(* CODESYS project SheetMetalFactoryLib.library
   Version: 0.0.0.1
   Author: RDOE
   Title: Sheet Metal Factory
   Description: Example Library to make use of FB Factory based on template provided with standard library project from wizard
   Placeholder: PlaceholderTemplate
   DocFormat: reStructuredText
   DefaultNamespace: SMF
   LanguageModelAttribute: qualified-access-only
   Company: OSB AG

Project tree, tasks and I/O mapping:
  libraries: CAA Types Extern, * (CAA Technical Workgroup); CAA Behaviour Model, * (CAA Technical Workgroup); CAA FB Factory, * (CAA Technical Workgroup)
  SheetMetalFactoryLib/
    Enums/
      data type ERROR
      data type WorkerDataType
      data type STATE
    Function Blocks/
      function block WorkerFactory [ST]: createIdle, prvInstCount, prvInstPoolExtendsFactor, prvInstSize, createCutter, createPolisher, createWorker
      function block ProcessController [ST]: FB_INIT
      Cutter/
        function block Cutter [ST]: init, prvInstInit, cutEdge, getState, setState, workerType, process, nextWorker, setNextWorker
        function block CutterData [ST]: workerType
      Polisher/
        function block Polisher [ST]: init, prvInstInit, polish, getState, setState, workerType, process, nextWorker, setNextWorker
        function block PolisherData [ST]: workerType
      Idle/
        function block Idle [ST]: setState, prvInstInit, nextWorker, workerType, process, setNextWorker
        function block IdleData [ST]: workerType
      function block SequenceFactory [ST]: FB_INIT, generateSequence, cleanUp
    Functions/
      Helper/
        function decrementInt [ST]
        function incrementInt [ST]
    GlobalConstants/
      global variables Constants
    GlobalVariables/
      global variables Variables
    Interfaces/
      interface IWorkerData: workerType
      interface IWorker: workerType, process, nextWorker, setNextWorker
    Structs/
    Templates/
      Behaviour Model/
        function block ETrigA_Temp [ST]: prvAbort, prvCyclicAction, prvResetOutputs, prvStart
        function block ETrigTlA_Temp [ST]: prvAbort, prvCyclicAction, prvResetOutputs, prvStart
        function block ETrigTl_Temp [ST]: prvAbort, prvCyclicAction, prvResetOutputs, prvStart
        function block ETrigToA_Temp [ST]: prvAbort, prvCyclicAction, prvResetOutputs, prvStart
        function block ETrigToTlA_Temp [ST]: prvAbort, prvCyclicAction, prvResetOutputs, prvStart
        function block ETrigToTl_Temp [ST]: prvAbort, prvCyclicAction, prvResetOutputs, prvStart
        function block ETrigTo_Temp [ST]: prvAbort, prvCyclicAction, prvResetOutputs, prvStart
        function block ETrig_Temp [ST]: prvAbort, prvCyclicAction, prvResetOutputs, prvStart
        function block LTrig_Temp [ST]: prvAbort, prvCyclicAction, prvResetOutputs, prvStart
      FB Factory/
        function block CustomData [ST]
        function block CustomFB [ST]: prvInstInit
        function block CustomFBFactory_heap [ST]: Create, prvInstCount, prvInstPoolExtendsFactor, prvInstSize
        function block CustomFBFactory_static [ST]: Create, prvInstPoolAdr, prvInstPoolSize, prvInstSize
    Types/
*)

// SheetMetalFactoryLib/Enums/ERROR
{attribute 'qualified_only'}
//{attribute 'conditionalshow'}
//{attribute 'conditionalshow' := 'SomeText'}
//{attribute 'hide'}
TYPE ERROR : 
(
	NO_ERROR := 0, 
	TIME_OUT
); 
END_TYPE

// SheetMetalFactoryLib/Enums/WorkerDataType
{attribute 'qualified_only'}
{attribute 'strict'}
TYPE WorkerDataType :
(
	NotSpecified :=-1,
	Idle := 0,
	Cutter,
	Polisher,
	Engraver
) := NotSpecified;
END_TYPE

// SheetMetalFactoryLib/Enums/STATE
{attribute 'qualified_only'}
{attribute 'strict'}
TYPE STATE :
(
	idle := 0,
	firstEdge,
	secondEdge,
	thirdEdge,
	fourthEdge,
	done,
	error := -1
	
);
END_TYPE

// SheetMetalFactoryLib/GlobalConstants/Constants
{attribute 'qualified_only'}
//{attribute 'conditionalshow'}
//{attribute 'conditionalshow' := 'SomeText'}
//{attribute 'hide'}
VAR_GLOBAL CONSTANT
	gc_iDummy : INT := 42; /// This is a dummy global constant variable
END_VAR

// SheetMetalFactoryLib/GlobalVariables/Variables
{attribute 'qualified_only'}
//{attribute 'conditionalshow'}
//{attribute 'conditionalshow' := 'SomeText'}
//{attribute 'hide'}
VAR_GLOBAL
	g_iDummy : INT; /// This is a dummy global variable
END_VAR

// SheetMetalFactoryLib/Templates/Behaviour Model/ETrigA_Temp
//{attribute 'hide_all_locals'}
//{attribute 'conditionalshow_all_locals' := 'SomeText'}
//{attribute 'conditionalshow_all_locals'}
//{attribute 'conditionalshow' := 'SomeText'}
//{attribute 'conditionalshow'}
//{attribute 'hide'}
FUNCTION_BLOCK ETrigA_Temp EXTENDS CBM.ETrigA
VAR_INPUT
	(* specific Inputs *)
END_VAR
VAR_OUTPUT
	eError : ERROR;
	(* specific Outputs *)
END_VAR
VAR
	(* specific vars *)
END_VAR

SUPER^();
IF iError = CBM.ERROR.TIME_OUT THEN
	eError := ERROR.TIME_OUT;
ELSE
	eError := iError;
END_IF

{attribute 'hide'}
METHOD prvAbort : BOOL
VAR_INPUT
END_VAR
VAR
END_VAR
IF xError THEN (* abort because of error *)
	(* TODO: insert specific Code here *)
ELSE (* user abort *)
	(* TODO: insert specific Code here *)
END_IF
xAbortInProgress:= FALSE;
END_METHOD

{attribute 'hide'}
METHOD prvCyclicAction : BOOL
VAR_INPUT
END_VAR
VAR
END_VAR
(* TODO: insert specific Code here *)
xDone:= TRUE;
(* if an error occurs, set iError to a value else than zero instead of xDone:= TRUE *)
(* to keep repeat loop *)
END_METHOD

{attribute 'hide'}
METHOD prvResetOutputs : BOOL
VAR_INPUT
END_VAR
VAR
END_VAR
(* TODO: insert specific Code here *)
SUPER^.prvResetOutputs();
END_METHOD

{attribute 'hide'}
METHOD prvStart : BOOL
VAR_INPUT
END_VAR
VAR
END_VAR
(* this code is called, when the application is started (rising edge of xExecute *)
(* TODO: copy specific input variables into local copies *)
(* TODO: insert specific Code here *)
;
END_METHOD

END_FUNCTION_BLOCK

// SheetMetalFactoryLib/Templates/Behaviour Model/ETrigTlA_Temp
//{attribute 'hide_all_locals'}
//{attribute 'conditionalshow_all_locals' := 'SomeText'}
//{attribute 'conditionalshow_all_locals'}
//{attribute 'conditionalshow' := 'SomeText'}
//{attribute 'conditionalshow'}
//{attribute 'hide'}
FUNCTION_BLOCK ETrigTlA_Temp EXTENDS CBM.ETrigTlA
VAR_INPUT
	(* specific Inputs *)
END_VAR
VAR_OUTPUT
	eError : ERROR;
	(* specific Outputs *)
END_VAR
VAR
	(* specific vars *)
END_VAR

SUPER^();
IF iError = CBM.ERROR.TIME_OUT THEN
	eError := ERROR.TIME_OUT;
ELSE
	eError := iError;
END_IF

{attribute 'hide'}
METHOD prvAbort : BOOL
VAR_INPUT
END_VAR
VAR
END_VAR
IF xError THEN (* abort because of error *)
	(* TODO: insert specific Code here *)
ELSE (* user abort *)
	(* TODO: insert specific Code here *)
END_IF
xAbortInProgress:= FALSE;
END_METHOD

{attribute 'hide'}
METHOD prvCyclicAction : BOOL
VAR_INPUT
END_VAR
VAR
END_VAR
(* TODO: insert specific Code here *)
xDone:= TRUE;
(* if an error occurs, set iError to a value else than zero instead of xDone:= TRUE *)
(* to keep repeat loop *)
END_METHOD

{attribute 'hide'}
METHOD prvResetOutputs : BOOL
VAR_INPUT
END_VAR
VAR
END_VAR
(* TODO: insert specific Code here *)
SUPER^.prvResetOutputs();
END_METHOD

{attribute 'hide'}
METHOD prvStart : BOOL
VAR_INPUT
END_VAR
VAR
END_VAR
(* this code is called, when the application is started (rising edge of xExecute *)
(* TODO: copy specific input variables into local copies *)
(* TODO: insert specific Code here *)
;
END_METHOD

END_FUNCTION_BLOCK

// SheetMetalFactoryLib/Templates/Behaviour Model/ETrigTl_Temp
//{attribute 'hide_all_locals'}
//{attribute 'conditionalshow_all_locals' := 'SomeText'}
//{attribute 'conditionalshow_all_locals'}
//{attribute 'conditionalshow' := 'SomeText'}
//{attribute 'conditionalshow'}
//{attribute 'hide'}
FUNCTION_BLOCK ETrigA_Temp EXTENDS CBM.ETrigTl
VAR_INPUT
	(* specific Inputs *)
END_VAR
VAR_OUTPUT
	eError : ERROR;
	(* specific Outputs *)
END_VAR
VAR
	(* specific vars *)
END_VAR

SUPER^();
IF iError = CBM.ERROR.TIME_OUT THEN
	eError := ERROR.TIME_OUT;
ELSE
	eError := iError;
END_IF

{attribute 'hide'}
METHOD prvAbort : BOOL
VAR_INPUT
END_VAR
VAR
END_VAR
IF xError THEN (* abort because of error *)
	(* TODO: insert specific Code here *)
ELSE (* user abort *)
	(* TODO: insert specific Code here *)
END_IF
xAbortInProgress:= FALSE;
END_METHOD

{attribute 'hide'}
METHOD prvCyclicAction : BOOL
VAR_INPUT
END_VAR
VAR
END_VAR
(* TODO: insert specific Code here *)
xDone:= TRUE;
(* if an error occurs, set iError to a value else than zero instead of xDone:= TRUE *)
(* to keep repeat loop *)
END_METHOD

{attribute 'hide'}
METHOD prvResetOutputs : BOOL
VAR_INPUT
END_VAR
VAR
END_VAR
(* TODO: insert specific Code here *)
SUPER^.prvResetOutputs();
END_METHOD

{attribute 'hide'}
METHOD prvStart : BOOL
VAR_INPUT
END_VAR
VAR
END_VAR
(* this code is called, when the application is started (rising edge of xExecute *)
(* TODO: copy specific input variables into local copies *)
(* TODO: insert specific Code here *)
;
END_METHOD

END_FUNCTION_BLOCK

// SheetMetalFactoryLib/Templates/Behaviour Model/ETrigToA_Temp
//{attribute 'hide_all_locals'}
//{attribute 'conditionalshow_all_locals' := 'SomeText'}
//{attribute 'conditionalshow_all_locals'}
//{attribute 'conditionalshow' := 'SomeText'}
//{attribute 'conditionalshow'}
//{attribute 'hide'}
FUNCTION_BLOCK ETrigToA_Temp EXTENDS CBM.ETrigToA
VAR_INPUT
	(* specific Inputs *)
END_VAR
VAR_OUTPUT
	eError : ERROR;
	(* specific Outputs *)
END_VAR
VAR
	(* specific vars *)
END_VAR

SUPER^();
IF iError = CBM.ERROR.TIME_OUT THEN
	eError := ERROR.TIME_OUT;
ELSE
	eError := iError;
END_IF

{attribute 'hide'}
METHOD prvAbort : BOOL
VAR_INPUT
END_VAR
VAR
END_VAR
IF xError THEN (* abort because of error *)
	(* TODO: insert specific Code here *)
ELSE (* user abort *)
	(* TODO: insert specific Code here *)
END_IF
xAbortInProgress:= FALSE;
END_METHOD

{attribute 'hide'}
METHOD prvCyclicAction : BOOL
VAR_INPUT
END_VAR
VAR
END_VAR
(* TODO: insert specific Code here *)
xDone:= TRUE;
(* if an error occurs, set iError to a value else than zero instead of xDone:= TRUE *)
END_METHOD

{attribute 'hide'}
METHOD prvResetOutputs : BOOL
VAR_INPUT
END_VAR
VAR
END_VAR
(* TODO: insert specific Code here *)
SUPER^.prvResetOutputs();
END_METHOD

{attribute 'hide'}
METHOD prvStart : BOOL
VAR_INPUT
END_VAR
VAR
END_VAR
(* this code is called, when the application is started (rising edge of xExecute *)
(* TODO: copy specific input variables into local copies *)
(* TODO: insert specific Code here *)
;
END_METHOD

END_FUNCTION_BLOCK

// SheetMetalFactoryLib/Templates/Behaviour Model/ETrigToTlA_Temp
//{attribute 'hide_all_locals'}
//{attribute 'conditionalshow_all_locals' := 'SomeText'}
//{attribute 'conditionalshow_all_locals'}
//{attribute 'conditionalshow' := 'SomeText'}
//{attribute 'conditionalshow'}
//{attribute 'hide'}
FUNCTION_BLOCK ETrigToTlA_Temp EXTENDS CBM.ETrigToTlA
VAR_INPUT
	(* specific Inputs *)
END_VAR
VAR_OUTPUT
	eError : ERROR;
	(* specific Outputs *)
END_VAR
VAR
	(* specific vars *)
END_VAR

SUPER^();
IF iError = CBM.ERROR.TIME_OUT THEN
	eError := ERROR.TIME_OUT;
ELSE
	eError := iError;
END_IF

{attribute 'hide'}
METHOD prvAbort : BOOL
VAR_INPUT
END_VAR
VAR
END_VAR
IF xError THEN (* abort because of error *)
	(* TODO: insert specific Code here *)
ELSE (* user abort *)
	(* TODO: insert specific Code here *)
END_IF
xAbortInProgress:= FALSE;
END_METHOD

{attribute 'hide'}
METHOD prvCyclicAction : BOOL
VAR_INPUT
END_VAR
VAR
END_VAR
(* TODO: insert specific Code here *)
xDone:= TRUE;
(* if an error occurs, set iError to a value else than zero instead of xDone:= TRUE *)
(* to keep repeat loop *)
END_METHOD

{attribute 'hide'}
METHOD prvResetOutputs : BOOL
VAR_INPUT
END_VAR
VAR
END_VAR
(* TODO: insert specific Code here *)
SUPER^.prvResetOutputs();
END_METHOD

{attribute 'hide'}
METHOD prvStart : BOOL
VAR_INPUT
END_VAR
VAR
END_VAR
(* this code is called, when the application is started (rising edge of xExecute *)
(* TODO: copy specific input variables into local copies *)
(* TODO: insert specific Code here *)
;
END_METHOD

END_FUNCTION_BLOCK

// SheetMetalFactoryLib/Templates/Behaviour Model/ETrigToTl_Temp
//{attribute 'hide_all_locals'}
//{attribute 'conditionalshow_all_locals' := 'SomeText'}
//{attribute 'conditionalshow_all_locals'}
//{attribute 'conditionalshow' := 'SomeText'}
//{attribute 'conditionalshow'}
//{attribute 'hide'}
FUNCTION_BLOCK ETrigToTl_Temp EXTENDS CBM.ETrigToTl
VAR_INPUT
	(* specific Inputs *)
END_VAR
VAR_OUTPUT
	eError : ERROR;
	(* specific Outputs *)
END_VAR
VAR
	(* specific vars *)
END_VAR

SUPER^();
IF iError = CBM.ERROR.TIME_OUT THEN
	eError := ERROR.TIME_OUT;
ELSE
	eError := iError;
END_IF

{attribute 'hide'}
METHOD prvAbort : BOOL
VAR_INPUT
END_VAR
VAR
END_VAR
IF xError THEN (* abort because of error *)
	(* TODO: insert specific Code here *)
ELSE (* user abort *)
	(* TODO: insert specific Code here *)
END_IF
xAbortInProgress:= FALSE;
END_METHOD

{attribute 'hide'}
METHOD prvCyclicAction : BOOL
VAR_INPUT
END_VAR
VAR
END_VAR
(* TODO: insert specific Code here *)
xDone:= TRUE;
(* if an error occurs, set iError to a value else than zero instead of xDone:= TRUE *)
(* to keep repeat loop *)
END_METHOD

{attribute 'hide'}
METHOD prvResetOutputs : BOOL
VAR_INPUT
END_VAR
VAR
END_VAR
(* TODO: insert specific Code here *)
SUPER^.prvResetOutputs();
END_METHOD

{attribute 'hide'}
METHOD prvStart : BOOL
VAR_INPUT
END_VAR
VAR
END_VAR
(* this code is called, when the application is started (rising edge of xExecute *)
(* TODO: copy specific input variables into local copies *)
(* TODO: insert specific Code here *)
;
END_METHOD

END_FUNCTION_BLOCK

// SheetMetalFactoryLib/Templates/Behaviour Model/ETrigTo_Temp
//{attribute 'hide_all_locals'}
//{attribute 'conditionalshow_all_locals' := 'SomeText'}
//{attribute 'conditionalshow_all_locals'}
//{attribute 'conditionalshow' := 'SomeText'}
//{attribute 'conditionalshow'}
//{attribute 'hide'}
FUNCTION_BLOCK ETrigTo_Temp EXTENDS CBM.ETrigTo
VAR_INPUT
	(* specific Inputs *)
END_VAR
VAR_OUTPUT
	eError : ERROR;
	(* specific Outputs *)
END_VAR
VAR
	(* specific vars *)
END_VAR

SUPER^();
IF iError = CBM.ERROR.TIME_OUT THEN
	eError := ERROR.TIME_OUT;
ELSE
	eError := iError;
END_IF

{attribute 'hide'}
METHOD prvAbort : BOOL
VAR_INPUT
END_VAR
VAR
END_VAR
IF xError THEN (* abort because of error *)
	(* TODO: insert specific Code here *)
ELSE (* user abort *)
	(* TODO: insert specific Code here *)
END_IF
xAbortInProgress:= FALSE;
END_METHOD

{attribute 'hide'}
METHOD prvCyclicAction : BOOL
VAR_INPUT
END_VAR
VAR
END_VAR
(* TODO: insert specific Code here *)
xDone:= TRUE;
(* if an error occurs, set iError to a value else than zero instead of xDone:= TRUE *)
(* to keep repeat loop *)
END_METHOD

{attribute 'hide'}
METHOD prvResetOutputs : BOOL
VAR_INPUT
END_VAR
VAR
END_VAR
(* TODO: insert specific Code here *)
SUPER^.prvResetOutputs();
END_METHOD

{attribute 'hide'}
METHOD prvStart : BOOL
VAR_INPUT
END_VAR
VAR
END_VAR
(* this code is called, when the application is started (rising edge of xExecute *)
(* TODO: copy specific input variables into local copies *)
(* TODO: insert specific Code here *)
;
END_METHOD

END_FUNCTION_BLOCK

// SheetMetalFactoryLib/Templates/Behaviour Model/ETrig_Temp
//{attribute 'hide_all_locals'}
//{attribute 'conditionalshow_all_locals' := 'SomeText'}
//{attribute 'conditionalshow_all_locals'}
//{attribute 'conditionalshow' := 'SomeText'}
//{attribute 'conditionalshow'}
//{attribute 'hide'}
FUNCTION_BLOCK ETrig_Temp EXTENDS CBM.ETrig
VAR_INPUT
	(* specific Inputs *)
END_VAR
VAR_OUTPUT
	eError : ERROR;
	(* specific Outputs *)
END_VAR
VAR
	(* specific vars *)
END_VAR

SUPER^();
IF iError = CBM.ERROR.TIME_OUT THEN
	eError := ERROR.TIME_OUT;
ELSE
	eError := iError;
END_IF

{attribute 'hide'}
METHOD prvAbort : BOOL
VAR_INPUT
END_VAR
VAR
END_VAR
IF xError THEN (* abort because of error *)
	(* TODO: insert specific Code here *)
ELSE (* user abort *)
	(* TODO: insert specific Code here *)
END_IF
xAbortInProgress:= FALSE;
END_METHOD

{attribute 'hide'}
METHOD prvCyclicAction : BOOL
VAR_INPUT
END_VAR
VAR
END_VAR
(* TODO: insert specific Code here *)
xDone:= TRUE;
(* if an error occurs, set iError to a value else than zero instead of xDone:= TRUE *)
(* to keep repeat loop *)
END_METHOD

{attribute 'hide'}
METHOD prvResetOutputs : BOOL
VAR_INPUT
END_VAR
VAR
END_VAR
(* TODO: insert specific Code here *)
SUPER^.prvResetOutputs();
END_METHOD

{attribute 'hide'}
METHOD prvStart : BOOL
VAR_INPUT
END_VAR
VAR
END_VAR
(* this code is called, when the application is started (rising edge of xExecute *)
(* TODO: copy specific input variables into local copies *)
(* TODO: insert specific Code here *)
;
END_METHOD

END_FUNCTION_BLOCK

// SheetMetalFactoryLib/Templates/Behaviour Model/LTrig_Temp
//{attribute 'hide_all_locals'}
//{attribute 'conditionalshow_all_locals' := 'SomeText'}
//{attribute 'conditionalshow_all_locals'}
//{attribute 'conditionalshow' := 'SomeText'}
//{attribute 'conditionalshow'}
//{attribute 'hide'}
FUNCTION_BLOCK LTrig_Temp EXTENDS CBM.LTrig
VAR_INPUT
	(* specific Inputs *)
END_VAR
VAR_OUTPUT
	eError : ERROR;
	(* specific Outputs *)
END_VAR
VAR
	(* specific vars *)
END_VAR

SUPER^();
IF iError = CBM.ERROR.TIME_OUT THEN
	eError := ERROR.TIME_OUT;
ELSE
	eError := iError;
END_IF

{attribute 'hide'}
METHOD prvAbort : BOOL
VAR_INPUT
END_VAR
VAR
END_VAR
IF xError THEN (* abort because of error *)
	(* TODO: insert specific Code here *)
ELSE (* user abort *)
	(* TODO: insert specific Code here *)
END_IF
xAbortInProgress:= FALSE;
END_METHOD

{attribute 'hide'}
METHOD prvCyclicAction : BOOL
VAR_INPUT
END_VAR
VAR
END_VAR
(* TODO: insert specific Code here *)
xDone:= TRUE;
(* if an error occurs, set iError to a value else than zero instead of xDone:= TRUE *)
(* to keep repeat loop *)
END_METHOD

{attribute 'hide'}
METHOD prvResetOutputs : BOOL
VAR_INPUT
END_VAR
VAR
END_VAR
(* TODO: insert specific Code here *)
SUPER^.prvResetOutputs();
END_METHOD

{attribute 'hide'}
METHOD prvStart : BOOL
VAR_INPUT
END_VAR
VAR
END_VAR
(* this code is called, when the application is started (rising edge of xExecute *)
(* TODO: copy specific input variables into local copies *)
(* TODO: insert specific Code here *)
;
END_METHOD

END_FUNCTION_BLOCK

// SheetMetalFactoryLib/Templates/FB Factory/CustomData
// This is a container to carry init data from the Create methode of the factory
// to the prvInstInit methode of the new generated function block instance
{attribute 'enable_dynamic_creation'}
//{attribute 'hide_all_locals'}
//{attribute 'conditionalshow_all_locals' := 'SomeText'}
//{attribute 'conditionalshow_all_locals'}
//{attribute 'conditionalshow' := 'SomeText'}
//{attribute 'conditionalshow'}
//{attribute 'hide'}
FUNCTION_BLOCK CustomData EXTENDS FBF.InstanceData
VAR_INPUT
	(* Todo: Add your application specific data as input variables *)
END_VAR

(* !! Do not add any executable code here !! *)
SUPER^();

END_FUNCTION_BLOCK

// SheetMetalFactoryLib/Templates/FB Factory/CustomFB
{attribute 'enable_dynamic_creation'}
//{attribute 'hide_all_locals'}
//{attribute 'conditionalshow_all_locals' := 'SomeText'}
//{attribute 'conditionalshow_all_locals'}
//{attribute 'conditionalshow' := 'SomeText'}
//{attribute 'conditionalshow'}
//{attribute 'hide'}
FUNCTION_BLOCK CustomFB EXTENDS FBF.InstanceBase;
VAR_INPUT
END_VAR
VAR_OUTPUT
END_VAR
VAR
END_VAR

SUPER^();

// This methode is called from the factory to give a chance
// to initialize the new fb instance with the content of itfData
//{attribute 'hide_all_locals'}
//{attribute 'conditionalshow_all_locals' := 'SomeText'}
//{attribute 'conditionalshow_all_locals'}
//{attribute 'conditionalshow' := 'SomeText'}
//{attribute 'conditionalshow'}
//{attribute 'hide'}
METHOD prvInstInit : FBF.ERROR
VAR_INPUT
	itfData : IData; 
END_VAR
VAR
	pData : POINTER TO CustomData;
	xOk : BOOL;
END_VAR
SUPER^.prvInstInit(itfData);
xOk := __QUERYPOINTER(itfData, pData);
IF xOk THEN
	(* THIS^.iLocalVar := pData^.iInitValue *);
END_IF
END_METHOD

END_FUNCTION_BLOCK

// SheetMetalFactoryLib/Templates/FB Factory/CustomFBFactory_heap
// This is a template for a factory with an heap based extendable memory pool
{attribute 'enable_dynamic_creation'}
//{attribute 'hide_all_locals'}
//{attribute 'conditionalshow_all_locals' := 'SomeText'}
//{attribute 'conditionalshow_all_locals'}
//{attribute 'conditionalshow' := 'SomeText'}
//{attribute 'conditionalshow'}
//{attribute 'hide'}
FUNCTION_BLOCK CustomFBFactory_heap EXTENDS FactoryBase
VAR
END_VAR

SUPER^();

(* Please replace CustonFB with your specific function block type *)
(* There is no need to change anything else !!! *)
METHOD Create : POINTER TO CustomFB
VAR_INPUT
	itfData : FBF.IData;
END_VAR
VAR_OUTPUT
	eError : FBF.ERROR;
END_VAR
VAR
	hInst : CAA.HANDLE;
	itfInst : FBF.IInstance;
	xOk : BOOL;
END_VAR
(* !!! This code must not be subject to change !!! *)
hInst := SUPER^.prvAllocInstMem(eError => eError);
Create := SUPER^.prvGetInstPointer(hInst);
IF Create <> 0 AND eError = FBF.ERROR.NO_ERROR THEN

	{implicit on}
	Create^.__vfInit();
	Create^.FB_Init(TRUE, FALSE);
	{implicit off}

	xOk := __QUERYINTERFACE(Create^, itfInst);
	IF xOk THEN
		xOk := SUPER^.prvInstInit(itfInst, hInst, itfData, eError=>eError);
	ELSE
		eError := FBF.ERROR.WRONG_INTERFACE;
	END_IF

	IF NOT xOk THEN
		SUPER^.prvFreeInstMem(hInst);
		Create := CAA.gc_pNULL;
	END_IF
END_IF
END_METHOD

//{attribute 'conditionalshow' := 'SomeText'}
//{attribute 'conditionalshow'}
//{attribute 'hide'}
PROPERTY prvInstCount : CAA.COUNT (* ctInst *)
GET
(* Please choose a proper value for prvInstCount *)
prvInstCount := 10;
END_GET
END_PROPERTY

//{attribute 'conditionalshow' := 'SomeText'}
//{attribute 'conditionalshow'}
//{attribute 'hide'}
PROPERTY prvInstPoolExtendsFactor : USINT (* usiFactor [0..x%] *)
GET
(* Please choose a proper value for prvInstPoolExtendsFactor *)
(* This value will be interpreted as a 0..x% size extendsion related to the original size of the pool *)
prvInstPoolExtendsFactor := 20;
END_GET
END_PROPERTY

//{attribute 'conditionalshow' := 'SomeText'}
//{attribute 'conditionalshow'}
//{attribute 'hide'}
PROPERTY prvInstSize : CAA.SIZE (* szInst *)
GET
(* Please replace CustomFB with your specific function block type *)
prvInstSize := sizeof(CustomFB);
END_GET
END_PROPERTY

END_FUNCTION_BLOCK

// SheetMetalFactoryLib/Templates/FB Factory/CustomFBFactory_static
// This is a template for a factory with an static iec memory based memory pool which a fixed capacity
{attribute 'enable_dynamic_creation'}
//{attribute 'hide_all_locals'}
//{attribute 'conditionalshow_all_locals' := 'SomeText'}
//{attribute 'conditionalshow_all_locals'}
//{attribute 'conditionalshow' := 'SomeText'}
//{attribute 'conditionalshow'}
//{attribute 'hide'}
FUNCTION_BLOCK CustomFBFactory_static EXTENDS FactoryBase
VAR
	// Please change the size of abyPoolMemory with your specific application need
	abyPoolMemory : ARRAY[0..529] OF BYTE;
END_VAR

SUPER^();

(* Please replace CustonFB with our specific function block type *)
(* There is no need to change anything else !!! *)
METHOD Create : POINTER TO CustomFB
VAR_INPUT
	itfData : FBF.IData;
END_VAR
VAR_OUTPUT
	eError : FBF.ERROR;
END_VAR
VAR
	hInst : CAA.HANDLE;
	itfInst : FBF.IInstance;
	xOk : BOOL;
END_VAR
(* !!! This code must not be subject to change !!! *)
hInst := SUPER^.prvAllocInstMem(eError => eError);
Create := SUPER^.prvGetInstPointer(hInst);
IF Create <> 0 AND eError = FBF.ERROR.NO_ERROR THEN

	{implicit on}
	Create^.__vfInit();
	Create^.FB_Init(TRUE, FALSE);
	{implicit off}

	xOk := __QUERYINTERFACE(Create^, itfInst);
	IF xOk THEN
		xOk := SUPER^.prvInstInit(itfInst, hInst, itfData, eError=>eError);
	ELSE
		eError := FBF.ERROR.WRONG_INTERFACE;
	END_IF

	IF NOT xOk THEN
		SUPER^.prvFreeInstMem(hInst);
		Create := CAA.gc_pNULL;
	END_IF
END_IF
END_METHOD

//{attribute 'conditionalshow' := 'SomeText'}
//{attribute 'conditionalshow'}
//{attribute 'hide'}
PROPERTY prvInstPoolAdr : CAA.PVOID (* pPool *)
GET
prvInstPoolAdr := ADR(abyPoolMemory);
END_GET
END_PROPERTY

//{attribute 'conditionalshow' := 'SomeText'}
//{attribute 'conditionalshow'}
//{attribute 'hide'}
PROPERTY prvInstPoolSize : CAA.SIZE (* szPool *)
GET
prvInstPoolSize := sizeof(abyPoolMemory);
END_GET
END_PROPERTY

//{attribute 'conditionalshow' := 'SomeText'}
//{attribute 'conditionalshow'}
//{attribute 'hide'}
PROPERTY prvInstSize : CAA.SIZE (* szInst *)
GET
(* Please replace CustomFB with your specific function block type *)
prvInstSize := sizeof(CustomFB);
END_GET
END_PROPERTY

END_FUNCTION_BLOCK

// SheetMetalFactoryLib/Function Blocks/Cutter/Cutter
{attribute 'enable_dynamic_creation'}
//{attribute 'hide_all_locals'}
//{attribute 'conditionalshow_all_locals' := 'SomeText'}
//{attribute 'conditionalshow_all_locals'}
//{attribute 'conditionalshow' := 'SomeText'}
//{attribute 'conditionalshow'}
//{attribute 'hide'}
FUNCTION_BLOCK Cutter EXTENDS FBF.InstanceBase IMPLEMENTS IWorker;
VAR_INPUT
END_VAR
VAR_OUTPUT
END_VAR
VAR
	_workerType : WorkerDataType;
	_nextWorker : IWorker;
	
	state : INT;
	
	xStart : DINT;
	yStart : DINT;
	xStop : DINT;
	yStop : DINT;
	
	xAct, xStep : DINT;
	yAct, yStep : DINT;
	
	_timeOfLastStep : TIME := T#0MS;
END_VAR
VAR CONSTANT
	STEPS : INT := 5;
	STEPTIME : TIME := T#100MS;

	STATE_ERROR : INT := -1;
	STATE_IDLE : INT := 0;
	STATE_BUSY : INT := 1;
	STATE_FIRST_EDGE : INT := 2;
	STATE_SECOND_EDGE : INT := 3;
	STATE_THIRD_EDGE : INT := 4;
	STATE_FOURTH_EDGE : INT := 5;
	STATE_DONE : INT := 6;

	SUCCESS : INT := 0;
END_VAR

SUPER^();

METHOD init
VAR_INPUT
END_VAR
THIS^.xAct := THIS^.xStart;
THIS^.yAct := THIS^.yStart;

THIS^.xStep := (THIS^.xStop - THIS^.xStart)/THIS^.STEPS;
THIS^.yStep := (THIS^.yStop - THIS^.yStart)/THIS^.STEPS;

THIS^.state := STATE_IDLE;
END_METHOD

// This methode is called from the factory to give a chance
// to initialize the new fb instance with the content of itfData
//{attribute 'hide_all_locals'}
//{attribute 'conditionalshow_all_locals' := 'SomeText'}
//{attribute 'conditionalshow_all_locals'}
//{attribute 'conditionalshow' := 'SomeText'}
//{attribute 'conditionalshow'}
//{attribute 'hide'}
METHOD prvInstInit : FBF.ERROR
VAR_INPUT
	itfData : FBF.IData; 
END_VAR
VAR
	pData : POINTER TO CutterData;
	xOk : BOOL;
END_VAR
SUPER^.prvInstInit(itfData);
xOk := __QUERYPOINTER(itfData, pData);
IF xOk THEN	
	THIS^._workerType := pData^.workerType;

	THIS^.xStart	:= REAL_TO_DINT(pData^.coords[0]*1000);
	THIS^.yStart 	:= REAL_TO_DINT(pData^.coords[1]*1000);
	THIS^.xStop 	:= REAL_TO_DINT(pData^.coords[2]*1000);
	THIS^.yStop 	:= REAL_TO_DINT(pData^.coords[3]*1000);
	
	THIS^.init();
END_IF
END_METHOD

METHOD cutEdge : int
VAR_INPUT
END_VAR
CASE getState() OF
	// 1st Edge
	STATE_FIRST_EDGE:
		IF (THIS^.xAct <> THIS^.xStop) THEN
			THIS^.xAct := THIS^.xAct + THIS^.xStep;
		ELSE
			setState(STATE_SECOND_EDGE);
		END_IF
 	// 2nd Edge
	STATE_SECOND_EDGE:
		IF (THIS^.yAct <> THIS^.yStop) THEN
			THIS^.yAct := THIS^.yAct + THIS^.yStep;
		ELSE
			setState(STATE_THIRD_EDGE);
		END_IF
	// 3rd Edge
	STATE_THIRD_EDGE:
		IF (THIS^.xAct <> THIS^.xStart) THEN
			THIS^.xAct := THIS^.xAct - THIS^.xStep;
		ELSE
			setState(STATE_FOURTH_EDGE);
		END_IF
	// 4th Edge
	STATE_FOURTH_EDGE:
		IF (THIS^.yAct <> THIS^.yStart) THEN
			THIS^.yAct := THIS^.yAct - THIS^.yStep;
		ELSE
			setState(STATE_DONE);
		END_IF
ELSE
	setState(STATE_ERROR);		
END_CASE

cutEdge := THIS^.getState();
END_METHOD

METHOD getState : INT
VAR_INPUT
END_VAR
getState := this^.state;
END_METHOD

METHOD setState
VAR_INPUT
	newState : INT;
END_VAR
this^.state := newState;
END_METHOD

PROPERTY workerType : WorkerDataType
GET
workerType := THIS^._workerType;
END_GET
END_PROPERTY

METHOD process : IWorker
VAR_INPUT
END_VAR
VAR
END_VAR
IF getState() = STATE_IDLE THEN
	setState(STATE_FIRST_EDGE);
END_IF

IF (TIME() - THIS^._timeOfLastStep) > STEPTIME THEN
	THIS^.cutEdge();
	THIS^._timeOfLastStep := TIME();
END_IF  


IF getState() = STATE_DONE THEN
	process := THIS^.nextWorker;
ELSE
	process := THIS^;	
END_IF
END_METHOD

PROPERTY nextWorker : IWorker
GET
nextWorker := this^._nextWorker;
END_GET
END_PROPERTY

METHOD setNextWorker : BOOL
VAR_INPUT
	nextWorker : IWorker;
END_VAR
THIS^._nextWorker := nextWorker;
END_METHOD

END_FUNCTION_BLOCK

// SheetMetalFactoryLib/Interfaces/IWorker
INTERFACE IWorker extends fbf.IInstance

PROPERTY workerType : WorkerDataType
GET
END_GET
END_PROPERTY

METHOD process : IWorker
VAR_INPUT
END_VAR
END_METHOD

PROPERTY nextWorker : IWorker
GET
END_GET
END_PROPERTY

METHOD setNextWorker : BOOL
VAR_INPUT
	nextWorker : IWorker;
END_VAR
END_METHOD

END_INTERFACE

// SheetMetalFactoryLib/Function Blocks/Cutter/CutterData
// This is a container to carry init data from the Create methode of the factory
// to the prvInstInit methode of the new generated function block instance
{attribute 'enable_dynamic_creation'}
//{attribute 'hide_all_locals'}
//{attribute 'conditionalshow_all_locals' := 'SomeText'}
//{attribute 'conditionalshow_all_locals'}
//{attribute 'conditionalshow' := 'SomeText'}
//{attribute 'conditionalshow'}
//{attribute 'hide'}
FUNCTION_BLOCK CutterData EXTENDS FBF.InstanceData IMPLEMENTS IWorkerData
VAR_INPUT
	coords : ARRAY [0..3] OF REAL;
	(*xStart : REAL;
	yStart : REAL;
	xStop : REAL;
	yStop : REAL;*)
END_VAR
VAR CONSTANT
	_workerType: WorkerDataType := WorkerDataType.Cutter;
END_VAR

(* !! Do not add any executable code here !! *)
SUPER^();

PROPERTY workerType : WorkerDataType
GET
workerType := this^._workerType;
END_GET
END_PROPERTY

END_FUNCTION_BLOCK

// SheetMetalFactoryLib/Interfaces/IWorkerData
INTERFACE IWorkerData EXTENDS FBF.IData

PROPERTY workerType : WorkerDataType
GET
END_GET
END_PROPERTY

END_INTERFACE

// SheetMetalFactoryLib/Function Blocks/WorkerFactory
// This is a template for a factory with an heap based extendable memory pool
{attribute 'enable_dynamic_creation'}
//{attribute 'hide_all_locals'}
//{attribute 'conditionalshow_all_locals' := 'SomeText'}
//{attribute 'conditionalshow_all_locals'}
//{attribute 'conditionalshow' := 'SomeText'}
//{attribute 'conditionalshow'}
//{attribute 'hide'}
FUNCTION_BLOCK WorkerFactory EXTENDS FBF.FactoryBase
VAR
END_VAR

SUPER^();

(* Please replace CustonFB with your specific function block type *)
(* There is no need to change anything else !!! *)
METHOD createIdle : POINTER TO Idle
VAR_INPUT
	itfData : FBF.IData;
END_VAR
VAR_OUTPUT
	eError : FBF.ERROR;
END_VAR
VAR
	hInst : CAA.HANDLE;
	itfInst : FBF.IInstance;
	xOk : BOOL;
END_VAR
(* !!! This code must not be subject to change !!! *)
hInst := SUPER^.prvAllocInstMem(eError => eError);
createIdle := SUPER^.prvGetInstPointer(hInst);
IF createIdle <> 0 AND eError = FBF.ERROR.NO_ERROR THEN

	{implicit on}
	createIdle^.__vfInit();
	createIdle^.FB_Init(TRUE, FALSE);
	{implicit off}

	xOk := __QUERYINTERFACE(createIdle^, itfInst);
	IF xOk THEN
		xOk := SUPER^.prvInstInit(itfInst, hInst, itfData, eError=>eError);
	ELSE
		eError := FBF.ERROR.WRONG_INTERFACE;
	END_IF

	IF NOT xOk THEN
		SUPER^.prvFreeInstMem(hInst);
		createIdle := CAA.gc_pNULL;
	END_IF
END_IF
END_METHOD

//{attribute 'conditionalshow' := 'SomeText'}
//{attribute 'conditionalshow'}
//{attribute 'hide'}
PROPERTY prvInstCount : CAA.COUNT (* ctInst *)
GET
(* Please choose a proper value for prvInstCount *)
prvInstCount := 10;
END_GET
END_PROPERTY

//{attribute 'conditionalshow' := 'SomeText'}
//{attribute 'conditionalshow'}
//{attribute 'hide'}
PROPERTY prvInstPoolExtendsFactor : USINT (* usiFactor [0..x%] *)
GET
(* Please choose a proper value for prvInstPoolExtendsFactor *)
(* This value will be interpreted as a 0..x% size extendsion related to the original size of the pool *)
prvInstPoolExtendsFactor := 20;
END_GET
END_PROPERTY

//{attribute 'conditionalshow' := 'SomeText'}
//{attribute 'conditionalshow'}
//{attribute 'hide'}
PROPERTY prvInstSize : CAA.SIZE (* szInst *)
GET
(* Please replace CustomFB with your specific function block type *)
prvInstSize := sizeof(Cutter);
END_GET
END_PROPERTY

(* Please replace CustonFB with your specific function block type *)
(* There is no need to change anything else !!! *)
METHOD createCutter : POINTER TO Cutter
VAR_INPUT
	itfData : FBF.IData;
END_VAR
VAR_OUTPUT
	eError : FBF.ERROR;
END_VAR
VAR
	hInst : CAA.HANDLE;
	itfInst : FBF.IInstance;
	xOk : BOOL;
END_VAR
(* !!! This code must not be subject to change !!! *)
hInst := SUPER^.prvAllocInstMem(eError => eError);
createCutter := SUPER^.prvGetInstPointer(hInst);
IF createCutter <> 0 AND eError = FBF.ERROR.NO_ERROR THEN

	{implicit on}
	createCutter^.__vfInit();
	createCutter^.FB_Init(TRUE, FALSE);
	{implicit off}

	xOk := __QUERYINTERFACE(createCutter^, itfInst);
	IF xOk THEN
		xOk := SUPER^.prvInstInit(itfInst, hInst, itfData, eError=>eError);
	ELSE
		eError := FBF.ERROR.WRONG_INTERFACE;
	END_IF

	IF NOT xOk THEN
		SUPER^.prvFreeInstMem(hInst);
		createCutter := CAA.gc_pNULL;
	END_IF
END_IF
END_METHOD

(* Please replace CustonFB with your specific function block type *)
(* There is no need to change anything else !!! *)
METHOD createPolisher : POINTER TO Polisher
VAR_INPUT
	itfData : FBF.IData;
END_VAR
VAR_OUTPUT
	eError : FBF.ERROR;
END_VAR
VAR
	hInst : CAA.HANDLE;
	itfInst : FBF.IInstance;
	xOk : BOOL;
END_VAR
(* !!! This code must not be subject to change !!! *)
hInst := SUPER^.prvAllocInstMem(eError => eError);
createPolisher := SUPER^.prvGetInstPointer(hInst);
IF createPolisher <> 0 AND eError = FBF.ERROR.NO_ERROR THEN

	{implicit on}
	createPolisher^.__vfInit();
	createPolisher^.FB_Init(TRUE, FALSE);
	{implicit off}

	xOk := __QUERYINTERFACE(createPolisher^, itfInst);
	IF xOk THEN
		xOk := SUPER^.prvInstInit(itfInst, hInst, itfData, eError=>eError);
	ELSE
		eError := FBF.ERROR.WRONG_INTERFACE;
	END_IF

	IF NOT xOk THEN
		SUPER^.prvFreeInstMem(hInst);
		createPolisher := CAA.gc_pNULL;
	END_IF
END_IF
END_METHOD

METHOD createWorker : IWorker
VAR_INPUT
	workerData : IWorkerData;
END_VAR
VAR
	cutter : POINTER TO Cutter;
	polisher : POINTER TO Polisher;
	idle: POINTER TO Idle;
	//engraver : POINTER TO Engraver;
END_VAR
CASE workerData.workerType OF
	WorkerDataType.Cutter:
		cutter := THIS^.createCutter(itfData:=workerData);
		__QUERYINTERFACE(cutter^,createWorker);
	WorkerDataType.Polisher:
		polisher := THIS^.createPolisher(itfData:=workerData);
		__QUERYINTERFACE(polisher^,createWorker);
	WorkerDataType.Engraver:
	WorkerDataType.Idle:
		idle := THIS^.createIdle(itfData:=workerData);
		__QUERYINTERFACE(idle^,createWorker);
	WorkerDataType.NotSpecified:
ELSE
	// do nothing		
END_CASE
END_METHOD

END_FUNCTION_BLOCK

// SheetMetalFactoryLib/Function Blocks/Idle/Idle
FUNCTION_BLOCK Idle EXTENDS FBF.InstanceBase IMPLEMENTS IWorker
VAR_INPUT
END_VAR
VAR_OUTPUT
END_VAR
VAR
	_workerType : WorkerDataType;
	_nextWorker : IWorker;
	
	state : INT;
	
	idleWild : BOOL;
END_VAR
VAR CONSTANT
	STATE_ERROR : INT := -1;
	STATE_IDLE : INT := 0;
	STATE_BUSY : INT := 1;
	STATE_DONE : INT := 2;

	SUCCESS : INT := 0;
END_VAR

METHOD setState
VAR_INPUT
	newState : INT;
END_VAR
this^.state := newState;
END_METHOD

METHOD prvInstInit : FBF.ERROR (* eError *)
VAR_INPUT
	itfData	: FBF.IData;
END_VAR
VAR
	pData : POINTER TO IdleData;
	xOk : BOOL;
END_VAR
SUPER^.prvInstInit(itfData);
xOk := __QUERYPOINTER(itfData, pData);
IF xOk THEN
	THIS^._nextWorker := THIS^;	
	THIS^._workerType := pData^.workerType;
	
	THIS^.setState(THIS^.STATE_IDLE);
END_IF
END_METHOD

PROPERTY nextWorker : IWorker
GET
nextworker:=this^._nextWorker;
END_GET
END_PROPERTY

PROPERTY workerType : WorkerDataType
GET
workerType := this^._workerType;
END_GET
END_PROPERTY

METHOD process : IWorker
this^.idleWild := not this^.idleWild;
process := THIS^;
END_METHOD

METHOD setNextWorker : BOOL
VAR_INPUT
	nextWorker : IWorker;
END_VAR
THIS^._nextWorker := THIS^;
END_METHOD

END_FUNCTION_BLOCK

// SheetMetalFactoryLib/Function Blocks/Idle/IdleData
// This is a container to carry init data from the Create methode of the factory
// to the prvInstInit methode of the new generated function block instance
{attribute 'enable_dynamic_creation'}
//{attribute 'hide_all_locals'}
//{attribute 'conditionalshow_all_locals' := 'SomeText'}
//{attribute 'conditionalshow_all_locals'}
//{attribute 'conditionalshow' := 'SomeText'}
//{attribute 'conditionalshow'}
//{attribute 'hide'}
FUNCTION_BLOCK IdleData EXTENDS FBF.InstanceData IMPLEMENTS IWorkerData
VAR_INPUT
END_VAR
VAR CONSTANT
	_workerType: WorkerDataType := WorkerDataType.Idle;
END_VAR

(* !! Do not add any executable code here !! *)
SUPER^();

{warning 'Eigenschaftenimplementierung hinzufügen'}
PROPERTY workerType : WorkerDataType
GET
workerType := this^._workerType;
END_GET
END_PROPERTY

END_FUNCTION_BLOCK

// SheetMetalFactoryLib/Function Blocks/Polisher/Polisher
{attribute 'enable_dynamic_creation'}
//{attribute 'hide_all_locals'}
//{attribute 'conditionalshow_all_locals' := 'SomeText'}
//{attribute 'conditionalshow_all_locals'}
//{attribute 'conditionalshow' := 'SomeText'}
//{attribute 'conditionalshow'}
//{attribute 'hide'}
FUNCTION_BLOCK Polisher EXTENDS FBF.InstanceBase IMPLEMENTS IWorker;
VAR_INPUT
END_VAR
VAR_OUTPUT
END_VAR
VAR
	_workerType : WorkerDataType;
	_nextWorker : IWorker;
	
	state : INT;
	
	polishDuration : TIME;
	startTime : TIME := T#0MS;
	
	polishCounter : DWORD := 0;
	
	
	
END_VAR
VAR CONSTANT
	STATE_ERROR : INT := -1;
	STATE_IDLE : INT := 0;
	STATE_BUSY : INT := 1;
	STATE_DONE : INT := 2;

	SUCCESS : INT := 0;
END_VAR

SUPER^();

METHOD init
VAR_INPUT
END_VAR
THIS^.state := STATE_IDLE;
END_METHOD

// This methode is called from the factory to give a chance
// to initialize the new fb instance with the content of itfData
//{attribute 'hide_all_locals'}
//{attribute 'conditionalshow_all_locals' := 'SomeText'}
//{attribute 'conditionalshow_all_locals'}
//{attribute 'conditionalshow' := 'SomeText'}
//{attribute 'conditionalshow'}
//{attribute 'hide'}
METHOD prvInstInit : FBF.ERROR
VAR_INPUT
	itfData : FBF.IData; 
END_VAR
VAR
	pData : POINTER TO PolisherData;
	xOk : BOOL;
END_VAR
SUPER^.prvInstInit(itfData);
xOk := __QUERYPOINTER(itfData, pData);
IF xOk THEN
	THIS^._workerType := pData^.workerType;
	
	THIS^.polishDuration := INT_TO_TIME(REAL_TO_INT(pData^.polishDuration));
	
	THIS^.init();
END_IF
END_METHOD

METHOD polish : INT
VAR_INPUT
END_VAR
IF THIS^.startTime = T#0MS THEN
	THIS^.startTime := TIME();
	THIS^.setState(THIS^.STATE_BUSY);
END_IF

IF (TIME() - THIS^.startTime) < THIS^.polishDuration THEN
	THIS^.polishCounter := THIS^.polishCounter + 1;
ELSE
	THIS^.setState(THIS^.STATE_DONE);
END_IF
END_METHOD

METHOD getState : INT
VAR_INPUT
END_VAR
getState := this^.state;
END_METHOD

METHOD setState
VAR_INPUT
	newState : INT;
END_VAR
this^.state := newState;
END_METHOD

PROPERTY workerType : WorkerDataType
GET
workerType := THIS^._workerType;
END_GET
END_PROPERTY

METHOD process : IWorker
VAR_INPUT
END_VAR
VAR
	
END_VAR
THIS^.polish();

IF getState() = STATE_DONE THEN
	process := THIS^.nextWorker;
ELSE
	process := THIS^;	
END_IF
END_METHOD

PROPERTY nextWorker : IWorker
GET
nextWorker := this^._nextWorker;
END_GET
END_PROPERTY

METHOD setNextWorker : BOOL
VAR_INPUT
	nextWorker : IWorker;
END_VAR
THIS^._nextWorker := nextWorker;
END_METHOD

END_FUNCTION_BLOCK

// SheetMetalFactoryLib/Function Blocks/Polisher/PolisherData
// This is a container to carry init data from the Create methode of the factory
// to the prvInstInit methode of the new generated function block instance
{attribute 'enable_dynamic_creation'}
//{attribute 'hide_all_locals'}
//{attribute 'conditionalshow_all_locals' := 'SomeText'}
//{attribute 'conditionalshow_all_locals'}
//{attribute 'conditionalshow' := 'SomeText'}
//{attribute 'conditionalshow'}
//{attribute 'hide'}
FUNCTION_BLOCK PolisherData EXTENDS FBF.InstanceData IMPLEMENTS IWorkerData
VAR_INPUT
	polishDuration : REAL;		//ms
END_VAR
VAR CONSTANT
	_workerType: WorkerDataType := WorkerDataType.Polisher;
END_VAR

(* !! Do not add any executable code here !! *)
SUPER^();

{warning 'Eigenschaftenimplementierung hinzufügen'}
PROPERTY workerType : WorkerDataType
GET
workerType := this^._workerType;
END_GET
END_PROPERTY

END_FUNCTION_BLOCK

// SheetMetalFactoryLib/Function Blocks/ProcessController
FUNCTION_BLOCK ProcessController
VAR_INPUT
END_VAR
VAR_OUTPUT
END_VAR
VAR
	worker : IWorker;
END_VAR

worker := worker.process();

METHOD FB_Init : BOOL
VAR_INPUT
  bInitRetains : BOOL; // TRUE: the Retain-variables are initialized (reset warm / reset cold)
  bInCopyCode : BOOL;  // TRUE  the instance will be copied to the copy-code afterward (online change)
  firstWorker : IWorker;
END_VAR
this^.worker := firstWorker;
END_METHOD

END_FUNCTION_BLOCK

// SheetMetalFactoryLib/Function Blocks/SequenceFactory
FUNCTION_BLOCK SequenceFactory
VAR_INPUT
	
END_VAR
VAR_OUTPUT
END_VAR
VAR_IN_OUT
	_recipe : ARRAY[*] OF IWorkerData;
END_VAR
VAR
	_workerFactory : WorkerFactory;
	_firstWorker : IWorker;
END_VAR

METHOD FB_Init : BOOL
VAR_INPUT
  bInitRetains : BOOL; // TRUE: the Retain-variables are initialized (reset warm / reset cold)
  bInCopyCode : BOOL;  // TRUE  the instance will be copied to the copy-code afterward (online change)

END_VAR
END_METHOD

METHOD generateSequence : IWorker
VAR_INPUT
END_VAR
VAR_IN_OUT
	recipe : ARRAY[*] OF IWorkerData;
END_VAR
VAR
	ii : DINT;		//loop counter variable
	actWorker : IWorker;
	prevWorker : IWorker;
END_VAR
ii := UPPER_BOUND(recipe,1);

WHILE ii >= LOWER_BOUND(recipe,1) DO
	actWorker := THIS^._workerFactory.createWorker(workerData:=recipe[ii]);
	
	IF NOT(actWorker.workerType = WorkerDataType.Idle) THEN
		actWorker.setNextWorker(prevWorker);	
	END_IF
	
	prevWorker := actWorker;
	
	ii := ii -1;
END_WHILE

THIS^._firstWorker := actWorker;

generateSequence := THIS^._firstWorker;
END_METHOD

METHOD cleanUp : BOOL
VAR_INPUT
END_VAR
VAR
	actWorker : IWorker;
	nextWorker : IWorker;
END_VAR
actWorker := THIS^._firstWorker;
nextWorker := actWorker.nextWorker;

WHILE nextWorker <> actWorker DO
	actWorker.Dispose();
	actWorker := nextWorker;
	nextWorker := actWorker.nextWorker;
END_WHILE

actWorker.Dispose();
THIS^._firstWorker := 0;
END_METHOD

END_FUNCTION_BLOCK

// SheetMetalFactoryLib/Functions/Helper/decrementInt
FUNCTION decrementInt : bool
VAR_INPUT
	var2Decrement : REFERENCE TO INT;
END_VAR
VAR
END_VAR

IF var2Decrement > -32768 THEN
	var2Decrement := var2Decrement - 1;
END_IF

END_FUNCTION

// SheetMetalFactoryLib/Functions/Helper/incrementInt
FUNCTION incrementInt : bool
VAR_INPUT
	var2Increment : REFERENCE TO INT;
	
END_VAR
VAR
END_VAR

IF var2Increment < 16#7FFF THEN
	var2Increment := var2Increment + 1;
END_IF

END_FUNCTION
